// TIA Portal V20 export
DATA_BLOCK "Data_block_1"   // DB1
{ S7_Optimized_Access := 'TRUE' }
// stored: MemoryReserve 100
   VAR
      "A" : Bool;
      "B" : Bool;
      C : Bool;
   END_VAR
BEGIN
END_DATA_BLOCK
